Staubli VAL3: IOInterface.dtx

public bool bBasicIO1
public bool bBasicIO2
dio diValveOut[2]
  [0] = {link=ValveIO\valve1}
  [1] = {link=ValveIO\valve2}
